// TIA Portal V17 export
// export: Created 2025-03-05T08:02:30.776104Z, ExportSetting WithDefaults, DisplayName Totally Integrated Automation Portal, DisplayVersion V17 Update 8, DisplayName TIA Portal Openness, DisplayVersion V17 Update 8, DisplayName TIA Portal Version Control Interface, DisplayVersion V17, DisplayName SINAMICS Startdrive Advanced, DisplayVersion V17 SP2, DisplayName SINAMICS Startdrive G110M, G120, G120C, G120D, G120P, G115D, DisplayVersion V17 SP2, DisplayName SINAMICS Startdrive G130, G150, S120, S150, SINAMICS MV, S210, DisplayVersion V17 SP2, DisplayName STEP 7 Professional, DisplayVersion V17 Update 8, DisplayName SINUMERIK ONE STEP 7 Toolbox, DisplayVersion V17 Update 12, DisplayName SINUMERIK 840D sl STEP 7 Toolbox, DisplayVersion V17 Update 12, DisplayName STEP 7 Safety, DisplayVersion V17 Update 6, DisplayName WinCC Advanced, DisplayVersion V17 Update 8
TYPE "POWDER FEEDER PLC AUXILIAR"
// stored: IsFailsafeCompliant false
   STRUCT
      o_fCarrierGasSelect : Bool;   // 0 = Argon Selected, 1 = Nitrogen Selected
      o_fUnitSelect : Bool;   // 0 = Metric Units, 1 = SI
      i_fCarrierGasSelected_Line1 : Bool;   // 0 = Argon Selected, 1 = Nitrogen Selected
      i_fCarrierGasSelected_Line2 : Bool;   // 0 = Argon Selected, 1 = Nitrogen Selected
      i_fCarrierGasSelectedAux : Bool;
      i_fUnitSelected_Line1 : Bool;   // 0 = Metric Units, 1 = SI
      i_fUnitSelected_Line2 : Bool;   // 0 = Metric Units, 1 = SI
      i_fUnitSelectedAux : Bool;
      o_rCarriergasNominal_Line1 : Real;   // Carrier Gas Setpoint [NLPM] (0..16 NLPM)
      o_rCarriergasNominal_Line2 : Real;   // Carrier Gas Setpoint [NLPM] (0..16 NLPM)
      o_rDiskSpeedNominal_Line1 : Real;   // Disk Speed Setpoint [%] (0..100 %)
      o_rDiskSpeedNominal_Line2 : Real;   // Disk Speed Setpoint [%] (0..100 %)
      o_rStirrerSpeedNominal_Line1 : Real;   // Stirrer Speed Setpoint [%] (30 - 100%)
      o_rStirrerSpeedNominal_Line2 : Real;   // Stirrer Speed Setpoint [%] (30 - 100%)
      o_rHopperTempNominal_Line1 : Real;   // Hopper Temperature Setpoint [°C] (n/a for Twin 150 R1.0)
      o_rHopperTempNominal_Line2 : Real;   // Hopper Temperature Setpoint [°C] (n/a for Twin 150 R1.0)
      o_rLLlimitCarriergas_Line1 : Real;   // Carrier Gas Flow LL Limit [NLPM] (Absolute Value)
      o_rLLlimitCarriergas_Line2 : Real;   // Carrier Gas Flow LL Limit [NLPM] (Absolute Value)
      o_rLLlimitDiskSpeedNominal_Line1 : Real;   // Disk Speed LL Limit [%] (Absolute Value)
      o_rLLlimitDiskSpeedNominal_Line2 : Real;   // Disk Speed LL Limit [%] (Absolute Value)
      o_rLLlimitStirrerSpeedNominal_Line1 : Real;   // Stirrer Speed LL Limit [%] (Absolute Value)
      o_rLLlimitStirrerSpeedNominal_Line2 : Real;   // Stirrer Speed LL Limit [%] (Absolute Value)
      o_rLlimitCarriergas_Line1 : Real;   // Carrier Gas L Limit [NLPM] (Absolute Value)
      o_rLlimitCarriergas_Line2 : Real;   // Carrier Gas L Limit [NLPM] (Absolute Value)
      o_rLlimitDiskSpeedNominal_Line1 : Real;   // Disk Speed L Limit [%] (Absolute Value)
      o_rLlimitDiskSpeedNominal_Line2 : Real;   // Disk Speed L Limit [%] (Absolute Value)
      o_rLlimitStirrerSpeedNominal_Line1 : Real;   // Stirrer Speed L Limit [%] (Absolute Value)
      o_rLlimitStirrerSpeedNominal_Line2 : Real;   // Stirrer Speed L Limit [%] (Absolute Value)
      o_rHlimitCarriergas_Line1 : Real;   // Carrier Gas H Limit [NLPM] (Absolute Value)
      o_rHlimitCarriergas_Line2 : Real;   // Carrier Gas H Limit [NLPM] (Absolute Value)
      o_rHlimitDiskSpeedNominal_Line1 : Real;   // Disk Speed H Limit [%] (Absolute Value)
      o_rHlimitDiskSpeedNominal_Line2 : Real;   // Disk Speed H Limit [%] (Absolute Value)
      o_rHlimitStirrerSpeedNominal_Line1 : Real;   // Stirrer Speed H Limit [%] (Absolute Value)
      o_rHlimitStirrerSpeedNominal_Line2 : Real;   // Stirrer Speed H Limit [%] (Absolute Value)
      o_rHHlimitCarriergas_Line1 : Real;   // Carrier Gas HH Limit [NLPM] (Absolute Value)
      o_rHHlimitCarriergas_Line2 : Real;   // Carrier Gas HH Limit [NLPM] (Absolute Value)
      o_rHHlimitDiskSpeedNominal_Line1 : Real;   // Disk Speed HH Limit [%] (Absolute Value)
      o_rHHlimitDiskSpeedNominal_Line2 : Real;   // Disk Speed HH Limit [%] (Absolute Value)
      o_rHHlimitStirrerSpeedNominal_Line1 : Real;   // Stirrer Speed HH Limit [%] (Absolute Value)
      o_rHHlimitStirrerSpeedNominal_Line2 : Real;   // Stirrer Speed HH Limit [%] (Absolute Value)
      o_rHHlimitHopperTempNominal_Line1 : Real;   // Hopper Temperature HH Limit (ºC), (Absolute Value, N/a For Twin 150 R1.0)
      o_rHHlimitHopperTempNominal_Line2 : Real;   // Hopper Temperature HH Limit (ºC), (Absolute Value, N/a For Twin 150 R1.0)
      i_rCarriergasActual_Line1 : Real;   // Actual Value Carriergas Flow (NLPM)
      i_rCarriergasActual_Line2 : Real;   // Actual Value Carriergas Flow (NLPM)
      i_rDiskActual_Line1 : Real;   // Actual Value Disk Speed (%)
      i_rDiskActual_Line2 : Real;   // Actual Value Disk Speed (%)
      i_rStirrerActual_Line1 : Real;   // Actual Value Stirrer Speed (%)
      i_rStirrerActual_Line2 : Real;   // Actual Value Stirrer Speed (%)
      i_rFeedrateActual_Line1 : Real;   // N/A For Twin 150
      i_rFeedrateActual_Line2 : Real;   // N/A For Twin 150
      i_rHopperTempActual_Line1 : Real;   // Actual Value Hopper Temperature (ºC)
      i_rHopperTempActual_Line2 : Real;   // Actual Value Hopper Temperature (ºC)
      i_rHopperPressureActual_Line1 : Real;   // Actual Value Hopper Pressure (Bar)
      i_rHopperPressureActual_Line2 : Real;   // Actual Value Hopper Pressure (Bar)
   END_STRUCT;
END_TYPE
